(* IEC 61131-3 sources: repolevel_ST_code_completion/output/0121完整版本/repoeval_Command1/readful_result_history, 31 files *)

(* ---- FB_AirConComfortCommand_0.st ---- *)
FUNCTION_BLOCK PUBLIC FB_AirConComfortCommand IMPLEMENTS I_Command
VAR
	refAirConditioning : REFERENCE TO FB_AirConditioning;
END_VAR

METHOD Execute : BOOL
VAR
	isValid : BOOL;
END_VAR

isValid := __ISVALIDREF(refAirConditioning);

IF isValid THEN
	refAirConditioning.Activate();
	refAirConditioning.SetTemperature(20.0);
	Execute := TRUE;
ELSE
	Execute := FALSE;
END_IF
END_FUNCTION_BLOCK

(* ---- FB_AirConComfortCommand_1.st ---- *)
FUNCTION_BLOCK PUBLIC FB_AirConComfortCommand IMPLEMENTS I_Command
VAR
	refAirConditioning : REFERENCE TO FB_AirConditioning;
END_VAR

METHOD Execute : BOOL
VAR
	isValid : BOOL;
END_VAR

isValid := (refAirConditioning <> 0);

IF isValid THEN
  refAirConditioning.Activate();
  refAirConditioning.SetTemperature(20.0);
  Execute := TRUE;
ELSE
  Execute := FALSE;
END_IF
END_FUNCTION_BLOCK

(* ---- FB_AirConComfortCommand_2.st ---- *)
FUNCTION_BLOCK PUBLIC FB_AirConComfortCommand IMPLEMENTS I_Command
VAR
	refAirConditioning : REFERENCE TO FB_AirConditioning;
END_VAR

METHOD Execute : BOOL
VAR
	isValid : BOOL;
END_VAR

isValid := (refAirConditioning <> 0);

IF isValid THEN
 refAirConditioning^ .Activate();
 refAirConditioning^ .SetTemperature(20.0);
 Execute := TRUE;
ELSE
 Execute := FALSE;
END_IF
END_FUNCTION_BLOCK

(* ---- FB_AirConComfortCommand_3.st ---- *)
FUNCTION_BLOCK PUBLIC FB_AirConComfortCommand IMPLEMENTS I_Command
VAR
	refAirConditioning : REFERENCE TO FB_AirConditioning;
END_VAR

METHOD Execute : BOOL
VAR
	isValid : BOOL;
END_VAR

isValid := (refAirConditioning <> 0);

IF isValid THEN
refAirConditioning^.Activate();
refAirConditioning^.SetTemperature(20.0);
Execute := TRUE;
ELSE
Execute := FALSE;
END_IF
END_FUNCTION_BLOCK

(* ---- FB_AirConditioning_0.st ---- *)
FUNCTION_BLOCK PUBLIC FB_AirConditioning
VAR_OUTPUT
	bActive			: BOOL;
	lrTemperature	: LREAL;
END_VAR
VAR
    bIsInitialized : BOOL := FALSE;
    lrDefaultTemperature : LREAL := 22.0;
END_VAR

IF NOT bIsInitialized THEN
    bActive := FALSE;
    lrTemperature := lrDefaultTemperature;
    bIsInitialized := TRUE;
END_IF;

IF bActive THEN
    (* Logic for active air conditioning can be added here if needed *)
ELSE
    (* Logic for inactive air conditioning can be added here if needed *)
END_IF;
END_FUNCTION_BLOCK

(* ---- FB_AirConditioning_1.st ---- *)
FUNCTION_BLOCK PUBLIC FB_AirConditioning
VAR_OUTPUT
	bActive			: BOOL;
	lrTemperature	: LREAL;
END_VAR
VAR
    bIsInitialized : BOOL := FALSE;
    lrDefaultTemperature : LREAL := 22.0;
END_VAR

IF NOT bIsInitialized THEN
  bActive := FALSE;
  lrTemperature := lrDefaultTemperature;
  bIsInitialized := TRUE;
END_IF

IF bActive THEN
  (* Logic for active air conditioning can be added here if needed *)
ELSE
  (* Logic for inactive air conditioning can be added here if needed *)
END_IF
END_FUNCTION_BLOCK

(* ---- FB_AirConStandbyCommand_0.st ---- *)
FUNCTION_BLOCK PUBLIC FB_AirConStandbyCommand IMPLEMENTS I_Command
VAR
    refAirConditioning : REFERENCE TO FB_AirConditioning;
END_VAR

IF __ISVALIDREF(refAirConditioning) THEN
    refAirConditioning.bActive := FALSE;
END_IF
END_FUNCTION_BLOCK

(* ---- FB_AirConStandbyCommand_1.st ---- *)
FUNCTION_BLOCK FB_AirConStandbyCommand IMPLEMENTS I_Command
VAR
  refAirConditioning : REFERENCE TO FB_AirConditioning;
END_VAR

IF __ISVALIDREF(refAirConditioning) THEN
  refAirConditioning.bActive := FALSE;
END_IF
END_FB

(* ---- FB_CDPlayer_0.st ---- *)
FUNCTION_BLOCK PUBLIC FB_CDPlayer
VAR_OUTPUT
	bPlayerActive		: BOOL;
	byVolume			: BYTE;
	byTrack				: UINT;
END_VAR
VAR
    bInitialized        : BOOL := FALSE;
END_VAR

IF NOT bInitialized THEN
    bPlayerActive := FALSE;
    byVolume := 50; // Default volume level
    byTrack := 1;   // Default track number
    bInitialized := TRUE;
END_IF;

CASE bPlayerActive OF
    TRUE:
        // Player is active, maintain current state
        bPlayerActive := TRUE;
    FALSE:
        // Player is inactive, reset outputs
        byVolume := 0;
        byTrack := 0;
END_CASE;
END_FUNCTION_BLOCK

(* ---- FB_CDPlayer_1.st ---- *)
FUNCTION_BLOCK PUBLIC FB_CDPlayer
VAR_OUTPUT
  bPlayerActive		: BOOL;
  byVolume			: BYTE;
  byTrack				: UINT;
END_VAR
VAR
  bInitialized        : BOOL := FALSE;
END_VAR

IF NOT bInitialized THEN
  bPlayerActive := FALSE;
  byVolume := 50; // Default volume level
  byTrack := 1;   // Default track number
  bInitialized := TRUE;
END_IF

CASE bPlayerActive OF
  TRUE:
    // Player is active, maintain current state
    bPlayerActive := TRUE;
  FALSE:
    // Player is inactive, reset outputs
    byVolume := 0;
    byTrack := 0;
END_CASE;
END_FUNCTION_BLOCK

(* ---- FB_CDPlayer_2.st ---- *)
FUNCTION_BLOCK PUBLIC FB_CDPlayer
VAR_OUTPUT
 bPlayerActive		: BOOL;
 byVolume			: BYTE;
 byTrack				: UINT;
END_VAR
VAR
 bInitialized        : BOOL := FALSE;
END_VAR

IF NOT bInitialized THEN
 bPlayerActive := FALSE;
 byVolume := 50; // Default volume level
 byTrack := 1;   // Default track number
 bInitialized := TRUE;
END_IF

IF bPlayerActive THEN
 // Player is active, maintain current state
 bPlayerActive := TRUE;
ELSE
 // Player is inactive, reset outputs
 byVolume := 0;
 byTrack := 0;
END_IF;
END_FUNCTION_BLOCK

(* ---- FB_CDPlayer_3.st ---- *)
FUNCTION_BLOCK PUBLIC FB_CDPlayer
VAR_OUTPUT
bPlayerActive		: BOOL;
byVolume			: BYTE;
byTrack				: UINT;
END_VAR
VAR
bInitialized        : BOOL := FALSE;
END_VAR

IF NOT bInitialized THEN
bPlayerActive := FALSE;
byVolume := 50; // Default volume level
byTrack := 1;   // Default track number
bInitialized := TRUE;
END_IF

IF bPlayerActive THEN
// Player is active, maintain current state
// No action needed here; bPlayerActive is already TRUE
ELSE
// Player is inactive, reset outputs
byVolume := 0;
byTrack := 0;
END_IF;
END_FUNCTION_BLOCK

(* ---- FB_Lamp_0.st ---- *)
FUNCTION_BLOCK PUBLIC FB_Lamp
VAR_OUTPUT
	byLevel			: BYTE;
END_VAR
VAR
    byCurrentLevel : BYTE := 0;
END_VAR

IF byCurrentLevel <> byLevel THEN
    byCurrentLevel := byLevel;
END_IF
END_FUNCTION_BLOCK

(* ---- FB_LampSetLevelCommand_0.st ---- *)
FUNCTION_BLOCK PUBLIC FB_LampSetLevelCommand IMPLEMENTS I_Command
VAR
	refLamp		: REFERENCE TO FB_Lamp;
	byNewLevel	: BYTE;
END_VAR

METHOD Execute : BOOL
VAR
	isSuccessful : BOOL;
END_VAR

IF __ISVALIDREF(refLamp) THEN
	isSuccessful := refLamp.SetLevel(byNewLevel);
	Execute := isSuccessful;
ELSE
	Execute := FALSE;
END_IF
END_FUNCTION_BLOCK

(* ---- FB_LampSetLevelCommand_2.st ---- *)
FUNCTION_BLOCK PUBLIC FB_LampSetLevelCommand IMPLEMENTS I_Command
VAR
	refLamp		: REFERENCE TO FB_Lamp;
	byNewLevel	: BYTE;
END_VAR

METHOD Execute : BOOL
VAR
	isSuccessful : BOOL;
END_VAR

IF __ISVALIDREF(refLamp) THEN
  // Check if the SetLevel method is callable and valid
  IF refLamp.SetLevel(byNewLevel) THEN
    isSuccessful := TRUE;
    Execute := isSuccessful;
  ELSE
    isSuccessful := FALSE;
    Execute := isSuccessful;
  END_IF;
ELSE
  Execute := FALSE;
END_IF
END_FUNCTION_BLOCK

(* ---- FB_LampSetLevelCommand_3.st ---- *)
FUNCTION_BLOCK PUBLIC FB_LampSetLevelCommand IMPLEMENTS I_Command
VAR
	refLamp		: REFERENCE TO FB_Lamp;
	byNewLevel	: BYTE;
END_VAR

METHOD Execute : BOOL
VAR
	isSuccessful : BOOL;
END_VAR

IF __ISVALIDREF(refLamp) THEN
 // Directly assign the result of SetLevel to Execute
 IF refLamp.SetLevel(byNewLevel) THEN
  Execute := TRUE;
 ELSE
  Execute := FALSE;
 END_IF;
ELSE
 Execute := FALSE;
END_IF
END_FUNCTION_BLOCK

(* ---- FB_MusicPlayCommand_0.st ---- *)
FUNCTION_BLOCK PUBLIC FB_MusicPlayCommand IMPLEMENTS I_Command
VAR
    refCDPlayer : REFERENCE TO FB_CDPlayer;
END_VAR

METHOD Execute
VAR
END_VAR

IF (__ISVALIDREF(THIS^.refCDPlayer)) THEN
    THIS^.refCDPlayer.SetVolume(40);
    THIS^.refCDPlayer.SetTrack(1);
    THIS^.refCDPlayer.Start();
END_IF
END_FUNCTION_BLOCK

(* ---- FB_MusicPlayCommand_1.st ---- *)
FUNCTION_BLOCK PUBLIC FB_MusicPlayCommand IMPLEMENTS I_Command
VAR
    refCDPlayer : REFERENCE TO FB_CDPlayer;
END_VAR

METHOD Execute
VAR
END_VAR

IF (__ISVALIDREF(refCDPlayer)) THEN
  refCDPlayer.SetVolume(40);
  refCDPlayer.SetTrack(1);
  refCDPlayer.Start();
END_IF
END_FUNCTION_BLOCK

(* ---- FB_MusicStopCommand_0.st ---- *)
FUNCTION_BLOCK PUBLIC FB_MusicStopCommand IMPLEMENTS I_Command
VAR
	refCDPlayer : REFERENCE TO FB_CDPlayer;
END_VAR

METHOD Execute
VAR
	refCDPlayer : REFERENCE TO FB_CDPlayer;
END_VAR

IF (__ISVALIDREF(THIS^.refCDPlayer)) THEN
	THIS^.refCDPlayer.Stop();
END_IF
END_FUNCTION_BLOCK

(* ---- FB_MusicStopCommand_1.st ---- *)
FUNCTION_BLOCK PUBLIC FB_MusicStopCommand IMPLEMENTS I_Command
VAR
	refCDPlayer : REFERENCE TO FB_CDPlayer;
END_VAR

METHOD Execute
// Removed redundant re-declaration of refCDPlayer to fix the shadowing error.

IF (__ISVALIDREF(THIS^.refCDPlayer)) THEN
  THIS^.refCDPlayer.Stop();
END_IF
END_FUNCTION_BLOCK

(* ---- FB_Socket_0.st ---- *)
FUNCTION_BLOCK PUBLIC FB_Socket
VAR_OUTPUT
	bActive		: BOOL;
END_VAR
VAR
    bInitialized : BOOL := FALSE;
END_VAR

IF NOT bInitialized THEN
    bActive := FALSE;
    bInitialized := TRUE;
END_IF;
END_FUNCTION_BLOCK

(* ---- FB_Socket_2.st ---- *)
FUNCTION_BLOCK PUBLIC FB_Socket
VAR_OUTPUT
  bActive		: BOOL;
END_VAR
VAR
  bInitialized : BOOL := FALSE;
END_VAR

IF NOT bInitialized THEN
  bActive := FALSE;
  bInitialized := TRUE;
END_IF
END_FUNCTION_BLOCK

(* ---- FB_Socket_3.st ---- *)
FUNCTION_BLOCK PUBLIC FB_Socket
VAR_OUTPUT
 bActive		: BOOL;
END_VAR
VAR
 bInitialized : BOOL := FALSE;
END_VAR

METHOD PUBLIC Main : VOID
IF NOT bInitialized THEN
 bActive := FALSE;
 bInitialized := TRUE;
END_IF
END_METHOD
END_FUNCTION_BLOCK

(* ---- FB_SocketOffCommand_0.st ---- *)
FUNCTION_BLOCK PUBLIC FB_SocketOffCommand IMPLEMENTS I_Command
VAR
    refSocket : REFERENCE TO FB_Socket;
END_VAR

IF __ISVALIDREF(refSocket) THEN
    refSocket.Off();
END_IF
END_FUNCTION_BLOCK

(* ---- FB_SocketOffCommand_1.st ---- *)
FUNCTION_BLOCK PUBLIC FB_SocketOffCommand IMPLEMENTS I_Command
VAR
  refSocket : REFERENCE TO FB_Socket;
END_VAR

IF __ISVALIDREF(refSocket) THEN
  refSocket.Off();
END_IF
END_FUNCTION

(* ---- FB_SocketOnCommand_0.st ---- *)
FUNCTION_BLOCK PUBLIC FB_SocketOnCommand IMPLEMENTS I_Command
VAR
    refSocket : REFERENCE TO FB_Socket;
END_VAR

METHOD Execute
VAR
END_VAR
IF (__ISVALIDREF(THIS^.refSocket)) THEN
    THIS^.refSocket.bActive := TRUE;
END_IF
END_FUNCTION_BLOCK

(* ---- FB_SocketOnCommand_1.st ---- *)
FUNCTION_BLOCK PUBLIC FB_SocketOnCommand IMPLEMENTS I_Command
VAR
  refSocket : REFERENCE TO FB_Socket;
END_VAR

METHOD Execute
VAR
END_VAR
IF (__ISVALIDREF(refSocket)) THEN
  refSocket^.bActive := TRUE;
END_IF
END_FUNCTION_BLOCK

(* ---- FB_SocketOnCommand_2.st ---- *)
FUNCTION_BLOCK PUBLIC FB_SocketOnCommand IMPLEMENTS I_Command
VAR
 refSocket : REFERENCE TO FB_Socket;
END_VAR

METHOD Execute
VAR
END_VAR
IF (__ISVALIDREF(refSocket)) THEN
 refSocket^.bActive := TRUE;
END_IF
END_FUNCTION_BLOCK

(* ---- FB_SocketOnCommand_3.st ---- *)
FUNCTION_BLOCK PUBLIC FB_SocketOnCommand IMPLEMENTS I_Command
VAR
refSocket : REFERENCE TO FB_Socket;
END_VAR

METHOD Execute
VAR
END_VAR
IF (__ISVALIDREF(refSocket)) THEN
refSocket^.bActive := TRUE;
END_IF
END_FUNCTION_BLOCK

(* ---- FB_SwitchPanel_0.st ---- *)
FUNCTION_BLOCK PUBLIC FB_SwitchPanel
VAR_INPUT
	arrSwitch		: ARRAY[1..8] OF BOOL;
END_VAR
VAR
	aiCommand		: ARRAY[1..8] OF I_Command;
	arrRtrig		: ARRAY[1..8] OF R_TRIG;
	nIndex			: INT;
END_VAR

FOR nIndex := 1 TO 8 DO
	arrRtrig[nIndex](CLK := arrSwitch[nIndex]);
	IF arrRtrig[nIndex].Q THEN
		IF (aiCommand[nIndex] <> 0) THEN
			aiCommand[nIndex].Execute();
		END_IF
	END_IF
END_FOR
END_FUNCTION_BLOCK

(* ---- FB_SwitchPanel_1.st ---- *)
FUNCTION_BLOCK PUBLIC FB_SwitchPanel
VAR_INPUT
	arrSwitch		: ARRAY[1..8] OF BOOL;
END_VAR
VAR
	aiCommand		: ARRAY[1..8] OF I_Command;
	arrRtrig		: ARRAY[1..8] OF R_TRIG;
	nIndex			: INT;
END_VAR

FOR nIndex := 1 TO 8 DO
  arrRtrig[nIndex](CLK := arrSwitch[nIndex]);
  IF arrRtrig[nIndex].Q THEN
    aiCommand[nIndex].Execute(); // Execute method of the initialized function block
  END_IF
END_FOR
END_FUNCTION_BLOCK
